(* CODESYS project Logging.library
   Company: Ziga Javornik
   DefaultNamespace: ZigaLibs.Logging
   Version: 0.0.4.1
   Placeholder: ZigaLibs.Logging
   Author: Ziga Javornik
   Description: A library containing file/logging functionalities.
   Title: ZigaLibs.Logging

Project tree, tasks and I/O mapping:
  libraries: Tc2_Standard, 3.4.5.0 (Beckhoff Automation GmbH); Tc2_System, 3.6.4.0 (Beckhoff Automation GmbH); Tc2_Utilities, * (Beckhoff Automation GmbH); Tc3_Module, 3.4.5.0 (Beckhoff Automation GmbH); TcError, 0.2.2.0 (Roald87); ZigaLibs.Core, 0.0.3.7 (Ziga Javornik); ZigaLibs.File, 0.2.2.0 (Ziga Javornik); TcUnit, 1.3.1 (www.tcunit.org)
  GVLs/
  SOURCE/
    Logger/
      DUTs/
        data type E_LoggerState
        data type ST_FileInfo
        data type ST_LoggerConfiguration
        data type ST_LogLevelHeaders
      POUs/
        function block FB_Logger [ST]: AddTimestampIfValidAndNewLine, Configuration, Configure, EnqueueLogEntry, GetLocalSystemTimeAsString, GetLogEntriesArrayMaxIndex, GetLogName, LogDefault, LogError, LogInfo, LogWarning, Reset
        function block FB_LoggerConfigBuilder [ST]: Apply, Configuration, DeleteLogsAfter, FB_init, SetLogExtension, SetLogFileName, SetLogFilePath, SetNetId, SetRollingInterval, Start
        interface I_Logger: LogDefault, LogError, LogInfo, LogWarning, Reset
        interface I_LoggerConfig: Configuration, Configure
        interface I_LoggerConfigBuilder: Apply, DeleteLogsAfter, SetLogExtension, SetLogFileName, SetLogFilePath, SetNetId, SetRollingInterval
  TESTS/
    Test suites/
      function block FB_Logger_Tests [ST]: Cleanup, Test01_LogError, Test02_LogWarning, Test03_LogInfo, Test04_LogGeneric, Test05_LogConfiguration_RollingIntervalSetTo0_ExpectOnlyFileName, Test06_FileExtension_DotAddedAutomaticallyIfNotProvided, Test07_ConfigurationDoesNotChangeUntilApplyIsCalled
    program PRG_TESTS [ST]
*)

// SOURCE/Logger/DUTs/E_LoggerState
{attribute 'qualified_only'}
{attribute 'strict'}
TYPE E_LoggerState :
(
	IDLE,
	PREPARE_LOG,
	OPEN_FILE,
	WRITE_TO_FILE,
	CLOSE_FILE,
	ERROR
);
END_TYPE

// SOURCE/Logger/DUTs/ST_FileInfo
TYPE ST_FileInfo :
STRUCT
	Location	: Tc2_System.T_MaxString;
	Path		: Tc2_System.T_MaxString;
END_STRUCT
END_TYPE

// SOURCE/Logger/DUTs/ST_LoggerConfiguration
TYPE ST_LoggerConfiguration :
STRUCT
	NetId				: Tc2_System.T_AmsNetID;	// Logger net-id, where the file will be generated
	FileName			: Tc2_System.T_MaxString;	// Name of the file
	FilePath			: Tc2_System.T_MaxString;	// Path to the file location
	FileExtension		: Tc2_System.T_MaxString := '.txt';	// File extension, with or without the preceding dot, will be checked when logging
	LogLevelHeaders		: ST_LogLevelHeaders;	// Log level headers for each log severity
	DeleteAfterDays		: UINT;	// Deletes files after X-many days, or never if set to 0
	DeleteCheckInterval	: TIME := T#6H;	// Defines how offten the logger will check the folder to delete old logs
	RollingInterval		: UINT := 6; // Sets the rolling interval (in hours) - how offten new log file is created. If set to 0, a single file is created. Beware of DeleteCheckInterval, which will delete this file and you will lose these files in that case.
	IsValid				: BOOL;	// Will be true as soon as configuration is applied
END_STRUCT
END_TYPE

// SOURCE/Logger/DUTs/ST_LogLevelHeaders
TYPE ST_LogLevelHeaders :
STRUCT
	Error	: STRING := '<Error> ';
	Warning	: STRING := '<Warning> ';
	Info	: STRING := '<Info> ';
END_STRUCT
END_TYPE

// SOURCE/Logger/POUs/FB_Logger
FUNCTION_BLOCK FB_Logger EXTENDS FB_ErrorSource IMPLEMENTS I_Logger, I_LoggerConfig
VAR
	_fileHandler				: ZigaLibs_File.FB_FileHandler;
	_logEntries					: ARRAY[0..100] OF Tc2_System.T_MaxString;
	_lastLogEntry				: Tc2_System.T_MaxString;
	_logEntryIndex				: ZigaLibs_Core.T_ArrayIndexer;
	_state						: E_LoggerState;
	_localSystemTimeProvider	: ZigaLibs_Core.FB_LocalSystemTimeProvider;
	_localSystemTimeString		: Tc2_System.T_MaxString;
	_stringBuilder				: ZigaLibs_Core.FB_StringBuilder;
	_dateForLogName				: STRING;
	_logEntriesMaxIndex			: ZigaLibs_Core.T_ArrayIndexer;
	_currentFileName			: Tc2_System.T_MaxString;
	_varInfo					: ZigaLibs_Core.T_VarInfo;
END_VAR

VAR PERSISTENT
	_configBuilder : FB_LoggerConfigBuilder(THIS^);
END_VAR

_localSystemTimeProvider();
_localSystemTimeString := GetLocalSystemTimeAsString();


CASE _state OF 
	E_LoggerState.IDLE:
		IF _logEntries[0] <> '' THEN
			_lastLogEntry := _logEntries[0];
			IF AddTimestampIfValidAndNewLine(_lastLogEntry) THEN
				_state := E_LoggerState.PREPARE_LOG;
			END_IF		
		END_IF

		
	E_LoggerState.PREPARE_LOG:
		_currentFileName := THIS^.GetLogName();
		_state := E_LoggerState.OPEN_FILE;
		
	E_LoggerState.OPEN_FILE:
		IF NOT _fileHandler.File.IsOpened THEN
			_fileHandler.Open(
				path := Configuration.FilePath, 
				name := _currentFileName, 
				mode := ZigaLibs_File.E_FileOpenMode.TEXT_APPEND,
				netId := Configuration.NetId);
			RETURN;
		END_IF	
		
		// Error opening the file
		IF _fileHandler.Error THEN
			THIS^.GenericError.Message := 'An error has occurred when opening the file!';
			THIS^.GenericError.Source := THIS^.InstancePath;
			THIS^.AdsError := _fileHandler.AdsError;
			_state := E_LoggerState.ERROR;
			RETURN;
		END_IF
		
		_state := E_LoggerState.WRITE_TO_FILE;

	E_LoggerState.WRITE_TO_FILE:
		IF NOT _fileHandler.WriteLine(_lastLogEntry) THEN
			RETURN;
		END_IF
		
		// Error writing to the file
		IF _fileHandler.Error THEN
			THIS^.GenericError.Message := 'An error has occurred when writing to file!';
			THIS^.GenericError.Source := THIS^.InstancePath;
			THIS^.AdsError := _fileHandler.AdsError;
			_state := E_LoggerState.ERROR;
			RETURN;
		END_IF
		
		_logEntriesMaxIndex := THIS^.GetLogEntriesArrayMaxIndex();
		// Remove the last entry, which was removed.
		ZigaLibs_Core.ArrayHelper.ShiftDown(arr := _logEntries, _logEntries[0]);
		
		_state := E_LoggerState.CLOSE_FILE;
		
	E_LoggerState.CLOSE_FILE:
		IF NOT _fileHandler.Close() THEN
			RETURN;
		END_IF

		// Error closing file.
		IF _fileHandler.Error THEN
			THIS^.GenericError.Message := 'An error occured when closing the file!';
			THIS^.GenericError.Source := THIS^.InstancePath;
			THIS^.AdsError := _fileHandler.AdsError;
			_state := E_LoggerState.ERROR;
			RETURN;
		END_IF

		_state := E_LoggerState.IDLE;

	E_LoggerState.ERROR:
		THIS^.Error := TRUE;
		// Wait for reset to be called...
		
END_CASE

METHOD PROTECTED AddTimestampIfValidAndNewLine : BOOL
VAR_INPUT
	entry	: REFERENCE TO Tc2_System.T_MaxString;
END_VAR
VAR
	sb	: ZigaLibs_Core.FB_StringBuilder;
END_VAR
IF _localSystemTimeProvider.CurrentTime.IsValid THEN
	entry := sb.AddString(_localSystemTimeString)
	.AddString(': ')
	.AddString(entry)
	.AddString(ZigaLibs_Core.StringConstants.NewLine)
	.Create();
	AddTimestampIfValidAndNewLine := TRUE;
END_IF
END_METHOD

// Gets the logger configuration
{attribute 'monitoring':='call'}
PROPERTY Configuration : REFERENCE TO ST_LoggerConfiguration
GET
Configuration REF= _configBuilder.Configuration;
END_GET
END_PROPERTY

METHOD Configure : I_LoggerConfigBuilder
Configure := _configBuilder;
_configBuilder.Start();
END_METHOD

METHOD PROTECTED EnqueueLogEntry
VAR_INPUT
	entry	: Tc2_System.T_MaxString;
END_VAR

VAR
	index	: ZigaLibs_Core.T_ArrayIndexer;
	maxIndex	: ZigaLibs_Core.T_ArrayIndexer;
END_VAR
maxIndex := THIS^.GetLogEntriesArrayMaxIndex();
FOR index := 0 TO maxIndex BY 1 DO
	IF _logEntries[index] = '' THEN
		_logEntries[index] := entry;
		EXIT;
	END_IF
END_FOR
END_METHOD

METHOD PRIVATE GetLocalSystemTimeAsString : T_MaxString
VAR_INPUT
END_VAR
GetLocalSystemTimeAsString :=_localSystemTimeProvider
	.ConvertToString()
	.DateTime(
		dateSeperator := '.',
		fillWithZeros := TRUE,
		IncludeMilliseconds := FALSE,
		timeFormat := ZigaLibs_Core.E_TimeFormat.YYMMDD_HHMMSS,
		timeOfDaySeperator := ':');
END_METHOD

METHOD PRIVATE GetLogEntriesArrayMaxIndex : ZigaLibs_Core.T_ArrayIndexer
VAR_INPUT
END_VAR
GetLogEntriesArrayMaxIndex := ZigaLibs_Core.ArrayHelper.GetMaxIndex(_logEntries, _logEntries[0], 0);
END_METHOD

METHOD PRIVATE GetLogName : T_MaxString
VAR_INPUT
END_VAR
VAR_INST
	sDate 					: Tc2_System.T_MaxString;
	sFileName				: Tc2_System.T_MaxString;
	sb						: FB_StringBuilder;
	rollingIntervalReached	: Tc2_Standard.R_TRIG;
END_VAR
IF THIS^.Configuration.RollingInterval = 0 THEN
	GetLogName := Tc2_Standard.CONCAT(THIS^.Configuration.FileName, THIS^.Configuration.FileExtension);
	RETURN;
END_IF


rollingIntervalReached(CLK := (_localSystemTimeProvider.CurrentTime.Value.wHour MOD THIS^.Configuration.RollingInterval) = 0);

IF sFileName = '' OR rollingIntervalReached.Q THEN
	sDate := _localSystemTimeProvider
		.ConvertToString()
		.DateTime(
			timeFormat := ZigaLibs_Core.E_TimeFormat.YYMMDD,
			timeOfDaySeperator := '',
			dateSeperator := '',
			fillWithZeros := TRUE,
			IncludeMilliseconds := FALSE);
	
	GetLogName := sb.Reset()
		.AddString(Configuration.FileName)
		.AddString('_')
		.AddString(sDate)
		.AddString('_')
		.AddString(_localSystemTimeProvider.ConvertToString().Hour(fillWithZeros := TRUE))
		.AddString(Configuration.FileExtension)
		.Create();	
END_IF
END_METHOD

(* Logs the message without any additions.*)
METHOD LogDefault
VAR_INPUT
	message	: Tc2_System.T_MaxString;
END_VAR
THIS^.EnqueueLogEntry(message);
END_METHOD

(* Logs the message by adding the error header to the start.*)
METHOD LogError
VAR_INPUT
	message	: Tc2_System.T_MaxString;
END_VAR
VAR
	sb	: FB_StringBuilder;
END_VAR
THIS^.EnqueueLogEntry(
	sb.AddString(Configuration.LogLevelHeaders.Error)
		.AddString(message)
		.Create());
END_METHOD

(* Logs the message by adding the info header to the start.*)
METHOD LogInfo
VAR_INPUT
	message	: Tc2_System.T_MaxString;
END_VAR
VAR
	sb	: FB_StringBuilder;
END_VAR
THIS^.EnqueueLogEntry(
	sb.AddString(Configuration.LogLevelHeaders.Info)
		.AddString(message)
		.Create());
END_METHOD

(* Logs the message by adding the info header to the start.*)
METHOD LogWarning
VAR_INPUT
	message	: Tc2_System.T_MaxString;
END_VAR
VAR
	sb	: FB_StringBuilder;
END_VAR
THIS^.EnqueueLogEntry(
	sb.AddString(Configuration.LogLevelHeaders.Warning)
		.AddString(message)
		.Create());
END_METHOD

METHOD Reset
IF THIS^.Error THEN
	_fileHandler.Reset();
	THIS^.ResetError();
	_state := E_LoggerState.IDLE;
END_IF
END_METHOD

END_FUNCTION_BLOCK

// SOURCE/Logger/POUs/I_Logger
// Provides logger
INTERFACE I_Logger

// Logs the message without any additions.
METHOD LogDefault
VAR_INPUT
	message	: Tc2_System.T_MaxString;
END_VAR
END_METHOD

// Logs the message by adding the error header to the start.
METHOD LogError
VAR_INPUT
	message	: Tc2_System.T_MaxString;
END_VAR
END_METHOD

// Logs the message by adding the info header to the start.
METHOD LogInfo
VAR_INPUT
	message	: Tc2_System.T_MaxString;
END_VAR
END_METHOD

// Logs the message by adding the info header to the start.
METHOD LogWarning
VAR_INPUT
	message	: Tc2_System.T_MaxString;
END_VAR
END_METHOD

METHOD Reset
VAR_INPUT
END_VAR
END_METHOD

END_INTERFACE

// SOURCE/Logger/POUs/I_LoggerConfig
INTERFACE I_LoggerConfig

// Gets the logger configuration - should not be edited, use .Configure() method to apply configuration.
{attribute 'monitoring':='call'}
PROPERTY Configuration : REFERENCE TO ST_LoggerConfiguration
GET
END_GET
END_PROPERTY

METHOD Configure : I_LoggerConfigBuilder
END_METHOD

END_INTERFACE

// SOURCE/Logger/POUs/I_LoggerConfigBuilder
INTERFACE I_LoggerConfigBuilder

// Applies the configuration
METHOD Apply
VAR_INPUT
	writeConfigToLog	: BOOL;	// Will write applied configuration to the target log file if set to TRUE
END_VAR
END_METHOD

(* Set the time after which the logs will be deleted.*)
METHOD DeleteLogsAfter : I_LoggerConfigBuilder
VAR_INPUT
	days			: UINT;	// Delete log files after X - days
	checkInterval	: TIME;	// Check interval for deleting the existing files
END_VAR
END_METHOD

(* Sets the log file extension <file>.<extension>. 
You can or can't include the dot, it will be checked and added either way.*)
METHOD SetLogExtension : I_LoggerConfigBuilder
VAR_INPUT
	extension	: STRING;
END_VAR
END_METHOD

// Sets the log file name
METHOD SetLogFileName : I_LoggerConfigBuilder
VAR_INPUT
	name	: STRING;
END_VAR
END_METHOD

// Sets the path where the logs will be stored.
METHOD SetLogFilePath : I_LoggerConfigBuilder
VAR_INPUT
	path	: Tc2_System.T_MaxString;
END_VAR
END_METHOD

// Sets the NetId of the device where logs will be stored.
METHOD SetNetId : I_LoggerConfigBuilder
VAR_INPUT
	netId	: Tc2_System.T_AmsNetID;
END_VAR
END_METHOD

// Sets the rolling interval (in hours) - how offten new log file is created. If set to 0, a single file is created. Beware of DeleteCheckInterval, which will delete this file and you will lose these files in that case.
METHOD SetRollingInterval : I_LoggerConfigBuilder
VAR_INPUT
	hours	: UINT;
END_VAR
END_METHOD

END_INTERFACE

// SOURCE/Logger/POUs/FB_LoggerConfigBuilder
FUNCTION_BLOCK FB_LoggerConfigBuilder IMPLEMENTS I_LoggerConfigBuilder
VAR_INPUT
END_VAR
VAR_OUTPUT
END_VAR
VAR
	_configuration 		: ST_LoggerConfiguration;
	_configurationTmp	: ST_LoggerConfiguration;
	_logger			: I_Logger;
END_VAR

(* Applies the configuration and returns I_Logger*)
METHOD Apply
VAR_INPUT
	writeConfigToLog	: BOOL;	// Will write applied configuration to the target log file if set to TRUE
END_VAR
VAR
	sb	: ZigaLibs_Core.FB_StringBuilder;
END_VAR
_configuration := _configurationTmp;
_configuration.IsValid := TRUE;

IF NOT writeConfigToLog THEN
	RETURN;
END_IF

// Too many string chains, CodeSys compiler crashes. Split to multiple lines.
_logger.LogDefault('==================== APPLYING LOGGER CONFIG ====================');
_logger.LogDefault(sb.Reset().AddString('NetId: ').AddString(_configuration.NetId).Create());
_logger.LogDefault(sb.Reset().AddString('File path: ').AddString(_configuration.FilePath).Create());
_logger.LogDefault(sb.Reset().AddString('File name: ').AddString(_configuration.FileName).Create());
_logger.LogDefault(sb.Reset().AddString('File extension: ').AddString(_configuration.FileExtension).Create());
_logger.LogDefault(sb.Reset().AddString('Delete after (days): ').addAny(_configuration.DeleteAfterDays).Create());
_logger.LogDefault(sb.Reset().AddString('Delete files check period: ').AddAny(_configuration.DeleteCheckInterval).Create());
_logger.LogDefault(sb.Reset().AddString('Error header: ').AddString(_configuration.LogLevelHeaders.Error).Create());
_logger.LogDefault(sb.Reset().AddString('Warning header: ').AddString(_configuration.LogLevelHeaders.Warning).Create());
_logger.LogDefault(sb.Reset().AddString('Info header: ').AddString(_configuration.LogLevelHeaders.Info).Create());
_logger.LogDefault('==================== LOGGER CONFIG APPLIED ====================');
END_METHOD

{attribute 'monitoring':='call'}
PROPERTY INTERNAL Configuration : REFERENCE TO ST_LoggerConfiguration
GET
Configuration REF= _configuration;
END_GET
END_PROPERTY

(* Set the time after which the logs will be deleted.*)
METHOD DeleteLogsAfter : I_LoggerConfigBuilder
VAR_INPUT
	days			: UINT;	// Delete log files after X - days
	checkInterval	: TIME;	// Check interval for deleting the existing files
END_VAR
_configurationTmp.DeleteAfterDays := days;
_configurationTmp.DeleteCheckInterval := checkInterval;
DeleteLogsAfter := THIS^;
END_METHOD

{attribute 'hide'}
METHOD FB_init : BOOL
VAR_INPUT
	bInitRetains : BOOL; // if TRUE, the retain variables are initialized (warm start / cold start)
	bInCopyCode : BOOL;  // if TRUE, the instance afterwards gets moved into the copy code (online change)
	logger	: I_Logger;
END_VAR
_logger := logger;
END_METHOD

(* Sets the log file extension <file>.<extension>. 
You can or can't include the dot, it will be checked and added either way.*)
METHOD SetLogExtension : I_LoggerConfigBuilder
VAR_INPUT
	extension	: STRING;
END_VAR
// Prepend the dot if it is not there already
IF Tc2_Standard.FIND(extension, '.') <> 1 THEN 
	extension := Tc2_Standard.CONCAT('.', extension);
END_IF
_configurationTmp.FileExtension := extension;
SetLogExtension := THIS^;
END_METHOD

(* Sets the log file name*)
METHOD SetLogFileName : I_LoggerConfigBuilder
VAR_INPUT
	name	: STRING;
END_VAR
_configurationTmp.FileName := name;
SetLogFileName := THIS^;
END_METHOD

(* Sets the path where the logs will be stored.*)
METHOD SetLogFilePath : I_LoggerConfigBuilder
VAR_INPUT
	path	: Tc2_System.T_MaxString;
END_VAR
_configurationTmp.FilePath := path;
SetLogFilePath := THIS^;
END_METHOD

(* Sets the NetId of the device where logs will be stored.*)
METHOD SetNetId : I_LoggerConfigBuilder
VAR_INPUT
	netId	: Tc2_System.T_AmsNetID;
END_VAR
_configurationTmp.NetId := netId;
SetNetId := THIS^;
END_METHOD

// Sets the rolling interval (in hours) - how offten new log file is created. If set to 0, a single file is created. Beware of DeleteCheckInterval, which will delete this file and you will lose these files in that case.
METHOD SetRollingInterval : I_LoggerConfigBuilder
VAR_INPUT
	hours	: UINT;
END_VAR
SetRollingInterval := THIS^;
_configurationTmp.RollingInterval := hours;
END_METHOD

// Shoould be called before any calls to configuration setting.
// This way temp configuration is equated to the current configuration.
// If some methods are not called, they will still have same values as oritinal configuration.
METHOD INTERNAL Start
_configurationTmp := _configuration;
END_METHOD

END_FUNCTION_BLOCK

// TESTS/Test suites/FB_Logger_Tests
FUNCTION_BLOCK INTERNAL FB_Logger_Tests EXTENDS FB_TestSuite
VAR
	_logger				: FB_Logger;
	_fileHandler		: ZigaLibs_File.FB_FileHandler;
	_localSystemTime	: ZigaLibs_Core.FB_LocalSystemTimeProvider;
	_loggerConfigured	: BOOL;
END_VAR

VAR CONSTANT
	FOLDER_PATH			: Tc2_System.T_MaxString 	:= '/home/Administrator/ZigaLibsTestFolder/LoggerTests/';
	NET_ID				: Tc2_System.T_AmsNetID 	:= '';
	LOG_NAME			: Tc2_System.T_MaxString 	:= 'MyLog';
	DATE_TIME_MAX_VALUE	: DT  := DATE_AND_TIME#2106-02-07-06:28:15;
END_VAR

// Configure logger...
IF NOT _loggerConfigured THEN
	_logger.Configure()
		.SetLogFilePath(FOLDER_PATH)
		.SetLogFileName(LOG_NAME)
		.SetLogExtension('log')
		.SetRollingInterval(6)
		.SetNetId(NET_ID)
		.DeleteLogsAfter(1, T#1H)
		.Apply(FALSE); 
	_loggerConfigured := TRUE;
END_IF

_logger();
_localSystemTime();

	
Test01_LogError();
Test02_LogWarning();
Test03_LogInfo();
Test04_LogGeneric();
Test05_LogConfiguration_RollingIntervalSetTo0_ExpectOnlyFileName();
Test06_FileExtension_DotAddedAutomaticallyIfNotProvided();
Test07_ConfigurationDoesNotChangeUntilApplyIsCalled();
Cleanup();

METHOD Cleanup
VAR_INPUT
END_VAR
IF TcUnit.TEST_ORDERED('Cleanup') THEN
	IF ZigaLibs_File.Utilities.Directory.DeleteFilesCreatedBefore(
		path := FOLDER_PATH, 
		fileNameContains := '.log', 
		netId := '', 
		thresholdDate := DATE_TIME_MAX_VALUE)
	THEN
		TcUnit.TEST_FINISHED();
	END_IF
END_IF
END_METHOD

METHOD Test01_LogError
VAR_INST
	bExists						: BOOL;
	TonMaxDelayForFileToAppear	: TON := (PT :=T#2S);
	fbStringBuilder				: ZigaLibs_Core.FB_StringBuilder;
	sDateForLogName 			: Tc2_System.T_MaxString;
	sReadContent				: Tc2_System.T_MaxString;
	nLogErrorTestState			: UINT := 0;
END_VAR
IF TcUnit.TEST_ORDERED('Test01_LogError')THEN
	CASE nLogErrorTestState OF
		0: 
			_logger.LogError('Error text....');
			nLogErrorTestState := nLogErrorTestState + 1;
		
		1:	
			IF _logger.Error THEN
				AssertTrue(
					Condition := FALSE, 
					Message := 'Unexpected error occurred when creating the log.');
					TcUnit.TEST_FINISHED();
					RETURN;
			END_IF
			
			TonMaxDelayForFileToAppear(IN := TRUE);
			IF TonMaxDelayForFileToAppear.Q THEN
				IF ZigaLibs_File.Utilities.File.Exists(
						name := _logger._fileHandler.File.Name,
						path := _logger._fileHandler.File.Path,
						NetId := _logger._fileHandler.File.NetId,
						Exists => bExists) 
				THEN
					AssertTrue(Condition := bExists,
						Message := 'Log file was not created!');
					nLogErrorTestState := nLogErrorTestState + 1;
				END_IF
			END_IF
				
		2:
			IF NOT _fileHandler.File.IsOpened THEN
				_fileHandler.Open(
					name := _logger._fileHandler.File.Name,
					path := _logger._fileHandler.File.Path,
					NetId := _logger._fileHandler.File.NetId,
					mode := ZigaLibs_File.E_FileOpenMode.TEXT_READ_MUST_EXIST);
				RETURN;
			END_IF
			
			IF _fileHandler.Read(sReadContent) THEN
				AssertTrue(
					Condition := Tc2_Standard.FIND(sReadContent,_logger.Configuration.LogLevelHeaders.Error) <> 0,
					Message := 'Error header not found in the read content of the log file!');
				
				AssertTrue(
					Condition := Tc2_Standard.FIND(sReadContent, 'Error text....') <> 0,
					Message := 'Message provided to the log method was not found in the contents of the file!');
					
				nLogErrorTestState := nLogErrorTestState + 1;
			END_IF
			
		3:
			IF _fileHandler.Close() THEN
				nLogErrorTestState := nLogErrorTestState + 1;
			END_IF	
			
		4:	
			IF ZigaLibs_File.Utilities.File.Delete(
				name := _logger._fileHandler.File.Name,
				path := _logger._fileHandler.File.Path,
				NetId := _logger._fileHandler.File.NetId,) 
			THEN
				TcUnit.TEST_FINISHED();
			END_IF
	END_CASE
END_IF
END_METHOD

METHOD Test02_LogWarning
VAR_INPUT
END_VAR

VAR_INST
	bExists						: BOOL;
	TonMaxDelayForFileToAppear	: TON := (PT :=T#2S);
	fbStringBuilder				: ZigaLibs_Core.FB_StringBuilder;
	sDateForLogName 			: Tc2_System.T_MaxString;
	sReadContent				: Tc2_System.T_MaxString;
	nLogWarningTestState		: UINT := 0;
END_VAR
IF TcUnit.TEST_ORDERED('Test02_LogWarning') THEN
	CASE nLogWarningTestState OF
		0: 
			_logger.LogWarning('Warning text....');
			nLogWarningTestState := nLogWarningTestState + 1;
		1:	
			IF _logger.Error THEN
				AssertTrue(
					Condition := FALSE, 
					Message := 'Unexpected error occurred when creating the log.');
					TcUnit.TEST_FINISHED();
					RETURN;
			END_IF
			
			TonMaxDelayForFileToAppear(IN := TRUE);
			IF TonMaxDelayForFileToAppear.Q AND_THEN 
				ZigaLibs_File.Utilities.File.Exists(
					name := _logger._fileHandler.File.Name,
					path := _logger._fileHandler.File.Path,
					NetId := _logger._fileHandler.File.NetId,
					Exists => bExists) 
			THEN
				AssertTrue( 
					Condition := bExists,
					Message := 'Log file was not created!');
				nLogWarningTestState := nLogWarningTestState + 1;
			END_IF
				
		2:
			IF NOT _fileHandler.File.IsOpened THEN
				_fileHandler.Open(
					name := _logger._fileHandler.File.Name,
					path := _logger._fileHandler.File.Path,
					NetId := _logger._fileHandler.File.NetId,
					mode := ZigaLibs_File.E_FileOpenMode.TEXT_READ_MUST_EXIST);
				RETURN;
			END_IF
			
			IF _fileHandler.Read(sReadContent) THEN
				AssertTrue(
					Condition := Tc2_Standard.FIND(sReadContent, _logger.Configuration.LogLevelHeaders.Warning) <> 0,
					Message := 'Warning header not found in the read content of the log file!');
	
				AssertTrue(
					Condition := Tc2_Standard.FIND(sReadContent, 'Warning text....') <> 0,
					Message := 'Message provided to the log method was not found in the contents of the file!');
					
				nLogWarningTestState := nLogWarningTestState + 1;
			END_IF
			
		3:
			IF _fileHandler.Close() THEN
				nLogWarningTestState := nLogWarningTestState + 1;
			END_IF	
			
		4:	
			IF ZigaLibs_File.Utilities.File.Delete(
				name := _logger._fileHandler.File.Name,
				path := _logger._fileHandler.File.Path,
				NetId := _logger._fileHandler.File.NetId,) 
			THEN
				TcUnit.TEST_FINISHED();
			END_IF
	END_CASE
END_IF
END_METHOD

METHOD Test03_LogInfo
VAR_INPUT
END_VAR
VAR_INST
	bExists						: BOOL;
	TonMaxDelayForFileToAppear	: TON := (PT :=T#2S);
	fbStringBuilder				: ZigaLibs_Core.FB_StringBuilder;
	sDateForLogName 			: Tc2_System.T_MaxString;
	sReadContent				: STRING(1000);
	nLogInfoState				: UINT := 0;
END_VAR
IF TcUnit.TEST_ORDERED('Test03_LogInfo') THEN
	CASE nLogInfoState OF
		0: 
			_logger.LogInfo('Info text....');
			nLogInfoState := nLogInfoState + 1;
		1:	
			IF _logger.Error THEN
				AssertTrue(
					Condition := FALSE, 
					Message := 'Unexpected error occurred when creating the log.');
					TcUnit.TEST_FINISHED();
					RETURN;
			END_IF
			
			
			TonMaxDelayForFileToAppear(IN := TRUE);
			IF TonMaxDelayForFileToAppear.Q AND_THEN 
				ZigaLibs_File.Utilities.File.Exists(
					name := _logger._fileHandler.File.Name,
					path := _logger._fileHandler.File.Path,
					NetId := _logger._fileHandler.File.NetId,
					Exists => bExists) 
			THEN
				AssertTrue( 
					Condition := bExists,
					Message := 'Log file was not created!');
				nLogInfoState := nLogInfoState + 1;
			END_IF
				
		2:
			IF NOT _fileHandler.File.IsOpened THEN
				_fileHandler.Open(
					name := _logger._fileHandler.File.Name,
					path := _logger._fileHandler.File.Path,
					NetId := _logger._fileHandler.File.NetId,
					mode := ZigaLibs_File.E_FileOpenMode.TEXT_READ_MUST_EXIST);
				RETURN;
			END_IF
			
			IF _fileHandler.Read(sReadContent) THEN
				AssertTrue(
					Condition := Tc2_Standard.FIND(sReadContent, _logger.Configuration.LogLevelHeaders.Info) <> 0,
					Message := 'Info header not found in the read content of the log file!');
	
				AssertTrue(
					Condition := Tc2_Standard.FIND(sReadContent, 'Info text....') <> 0,
					Message := 'Message provided to the log method was not found in the contents of the file!');
					
				nLogInfoState := nLogInfoState + 1;
			END_IF
			
		3:
			IF _fileHandler.Close() THEN
				nLogInfoState := nLogInfoState + 1;
			END_IF	
			
		4:	
			IF ZigaLibs_File.Utilities.File.Delete(
				name := _logger._fileHandler.File.Name,
				path := _logger._fileHandler.File.Path,
				NetId := _logger._fileHandler.File.NetId,) 
			THEN
				TcUnit.TEST_FINISHED();
			END_IF
	END_CASE
END_IF
END_METHOD

METHOD Test04_LogGeneric
VAR_INST
	bExists						: BOOL;
	TonMaxDelayForFileToAppear	: TON := (PT :=T#2S);
	fbStringBuilder				: ZigaLibs_Core.FB_StringBuilder;
	sDateForLogName 			: Tc2_System.T_MaxString;
	sReadContent				: STRING(1000);
	nLogGenericState			: UINT := 0;
END_VAR
IF TcUnit.TEST_ORDERED('Test04_LogGeneric') THEN
	CASE nLogGenericState OF
		0: 
			_logger.LogDefault('Default text....');
			nLogGenericState := nLogGenericState + 1;
			
		1:	
			IF _logger.Error THEN
				AssertTrue(
					Condition := FALSE, 
					Message := 'Unexpected error occurred when creating the log.');
					TcUnit.TEST_FINISHED();
					RETURN;
			END_IF
			
			TonMaxDelayForFileToAppear(IN := TRUE);
			IF TonMaxDelayForFileToAppear.Q AND_THEN 
				ZigaLibs_File.Utilities.File.Exists(
					name := _logger._fileHandler.File.Name,
					path := _logger._fileHandler.File.Path,
					NetId := _logger._fileHandler.File.NetId,
					Exists => bExists) 
			THEN
				AssertTrue( 
					Condition := bExists,
					Message := 'Log file was not created!');
				nLogGenericState := nLogGenericState + 1;
			END_IF
				
		2:
			IF NOT _fileHandler.File.IsOpened THEN
				_fileHandler.Open(
					name := _logger._fileHandler.File.Name,
					path := _logger._fileHandler.File.Path,
					NetId := _logger._fileHandler.File.NetId,
					mode := ZigaLibs_File.E_FileOpenMode.TEXT_READ_MUST_EXIST);
				RETURN;
			END_IF
			
			IF _fileHandler.Read(sReadContent) THEN
				AssertFalse(
					Condition := Tc2_Standard.FIND(sReadContent, _logger.Configuration.LogLevelHeaders.Info) <> 0,
					Message := 'Info header was found in the read content of the log file!');
					
				AssertFalse(
					Condition := Tc2_Standard.FIND(sReadContent, _logger.Configuration.LogLevelHeaders.Warning) <> 0,
					Message := 'Warning header was found in the read content of the log file!');
				
				AssertFalse(
					Condition := Tc2_Standard.FIND(sReadContent, _logger.Configuration.LogLevelHeaders.Error) <> 0,
					Message := 'Error header was found in the read content of the log file!');
					
				AssertTrue(
					Condition := Tc2_Standard.FIND(sReadContent, 'Default text....') <> 0,
					Message := 'Default log message not found.');
					
				nLogGenericState := nLogGenericState + 1;
			END_IF
			
		3:
			IF _fileHandler.Close() THEN
				nLogGenericState := nLogGenericState + 1;
			END_IF	
			
		4:	
			IF ZigaLibs_File.Utilities.File.Delete(
				name := _logger._fileHandler.File.Name,
				path := _logger._fileHandler.File.Path,
				NetId := _logger._fileHandler.File.NetId,) 
			THEN
				TcUnit.TEST_FINISHED();
			END_IF
	END_CASE
END_IF
END_METHOD

METHOD Test05_LogConfiguration_RollingIntervalSetTo0_ExpectOnlyFileName
VAR_INPUT
END_VAR
VAR_INST
	step	: INT;
	fileExists	: BOOL;
END_VAR
IF TcUnit.TEST_ORDERED('Test05_LogConfiguration_RollingIntervalSetTo0_ExpectOnlyFileName') THEN
	CASE step OF
		0:	
			_logger.Configure()
				.SetRollingInterval(0)
				.Apply(FALSE);
			step := step + 1;
			
		1:
			_logger.LogInfo('test..');	
			step := step + 1;
			
		2:
			IF ZigaLibs_File.Utilities.File.Exists(
				FOLDER_PATH, 
				TC2_Standard.CONCAT(LOG_NAME, _logger.Configuration.FileExtension), 
				NET_ID, 
				result => fileExists) 
			THEN
				AssertTrue(fileExists, 'Setting rolling interval to 0, the expected file was not craeted.');
				step := step + 1;
			END_IF
			
		3:
			IF fileExists THEN
				IF ZigaLibs_File.Utilities.File.Delete(
					FOLDER_PATH, 
					TC2_Standard.CONCAT(LOG_NAME, _logger.Configuration.FileExtension), 
					NET_ID) 
				THEN
					TcUnit.TEST_FINISHED();	
				END_IF
			END_IF
	END_CASE
END_IF
END_METHOD

METHOD Test06_FileExtension_DotAddedAutomaticallyIfNotProvided
VAR_INPUT
END_VAR
IF TcUnit.TEST_ORDERED('Test06_FileExtension_DotAddedAutomaticallyIfNotProvided') THEN
	_logger.Configure().SetLogExtension('NoDotAdded').Apply(FALSE);
	AssertEquals_STRING(
		'.NoDotAdded',
		_logger.Configuration.FileExtension,
		'If no dot is prepended to the file extension, it should be added automatically.');
		
	_logger.Configure().SetLogExtension('.DotAdded').Apply(FALSE);
	AssertEquals_STRING(
		'.DotAdded',
		_logger.Configuration.FileExtension,
		'If dot is prepended to the file extension, it should not be added automatically as it already exists.');
	TcUnit.TEST_FINISHED();
END_IF
END_METHOD

METHOD Test07_ConfigurationDoesNotChangeUntilApplyIsCalled
VAR_INPUT
END_VAR
VAR
	originalConfiguration	: ST_LoggerConfiguration;
END_VAR
IF TcUnit.TEST_ORDERED('Test07_ConfigurationDoesNotChangeUntilApplyIsCalled') THEN
	originalConfiguration := _logger.Configuration;
	
	_logger.Configure().SetLogFileName('lalal');
	AssertEquals_STRING(originalConfiguration.FileName, _logger.Configuration.FileName,
		'Until apply is called, the configuration should not be applied.');
		
	_logger.Configure().SetLogFileName('test123').Apply(FALSE);
	AssertEquals_STRING('test123', _logger.Configuration.FileName,
		'When apply is called, the configuration should be applied.');
		
	TcUnit.TEST_FINISHED();
END_IF
END_METHOD

END_FUNCTION_BLOCK

// TESTS/PRG_TESTS
PROGRAM INTERNAL PRG_TESTS

(* Instantiate test suites here. Naming convention for tests should be a suffix with _Tests.
Good practice for creating test methods is to end them with _test as well. *)
VAR
	LoggerTests			: FB_Logger_Tests;
END_VAR

// Run tests in paralel
//TcUnit.RUN();

// Run tests in sequence, one after the other. Uncomment if required.
TcUnit.RUN_IN_SEQUENCE();

END_PROGRAM
